(* IEC 61131-3 sources: Stat_Resistant_AI_Coding/src/plc/project/Station010/SqS_Wp100_Run, 2 files *)

(* ---- declaration.st ---- *)
FUNCTION_BLOCK SqS_Wp100_Run EXTENDS OpconSfcChain
////<OES_INFO Mode="Merge" Areas="1/1" />
////<OES_CODE MergeId="Declaration">{{{
VAR_INPUT
  rUnit      : REFERENCE TO Wp100Unit;
  MeasurePos : MeasurePsoEnum;
END_VAR
////<END_OES_CODE>}}}

VAR_OUTPUT
  /// Result remains valid after DONE and is cleared when the next execution starts
  Result : Wp100RunResultStruct;
END_VAR

VAR
  _positionValid         : BOOL;
  _startButton           : MachineCommon.FB_OperatorButton;
  _safetyDoorCloseStarted : BOOL;
  _pressDownStarted      : BOOL;
  _kistlerStarted        : BOOL;
  _kistlerStopRequested  : BOOL;
  _bursterStarted        : BOOL;
  _pressUpStarted        : BOOL;
  _safetyDoorOpenStarted : BOOL;
  _pressDelay            : TON;
  _unitResult            : DINT;
END_VAR

(* ---- OnChainFinish.st ---- *)
/// Method is called for only one cycle if chain stops working by any given reason
METHOD PROTECTED OnChainFinish
VAR_INPUT
  Reason: OpconChainFinishReason;
END_VAR

// Call base method
// AI_HMI_FORCE_TRACE_BEGIN
CASE Reason OF
  OpconChainFinishReason.ERROR:
    Station.ForceTraceAddon.Recorder.Finish(Reason := 4,
      LastForceN := Wp100A104Kistler.Unit.OutImm.ForceAct);
  OpconChainFinishReason.CANCEL:
    Station.ForceTraceAddon.Recorder.Finish(Reason := 3,
      LastForceN := Wp100A104Kistler.Unit.OutImm.ForceAct);
END_CASE
// AI_HMI_FORCE_TRACE_END
SUPER^.OnChainFinish(Reason);

// A cancelled/finished SFC no longer calls its active action. Reset every
// request owned by this chain and leave the stored Result available to caller.
_startButton(
  Execute       := FALSE,
  ButtonPressed := FALSE,
  Blink500ms    := FALSE
);
BinIo._000P610 := _startButton.LampOn;

_pressDelay(IN := FALSE, PT := T#0MS);
_unitResult := CheckPressForce(Phase := 0);

AiWp100.BursterProgramSelect(
  Execute := FALSE,
  ProgramNo := 0
);
Wp100K101SafetyDoor.Unit.Execute       := FALSE;
Wp100K102PressingCylinder.Unit.Execute := FALSE;
Wp100A103ResistantDetector.Unit.Execute := FALSE;
// Execute's falling edge invokes the standard Unit Cancel. Do not issue an
// EndMeasurement request here: a preflight failure may never have started it.
Wp100A104Kistler.Unit.ParImm.EndMeasurement := FALSE;
Wp100A104Kistler.Unit.Execute := FALSE;
_unitResult := CheckKistlerProgram(Reset := TRUE);

_positionValid          := FALSE;
_safetyDoorCloseStarted := FALSE;
_pressDownStarted       := FALSE;
_kistlerStarted         := FALSE;
_kistlerStopRequested   := FALSE;
_bursterStarted         := FALSE;
_pressUpStarted         := FALSE;
_safetyDoorOpenStarted  := FALSE;

CASE Reason
OF
  OpconChainFinishReason.ERROR,
  OpconChainFinishReason.CANCEL:
    Station._AutoInfoline := AutoInfoLineEnum.USER_INFO_TEXT_CLEAR;

  OpconChainFinishReason.DONE:
    ; // N999 clears the atomic prompt; the parent chain owns the next prompt.

  ELSE
    ; // do nothing
END_CASE
